INTERFACE I_TestRunner

METHOD AddTest
VAR_INPUT
    UnitTest : I_UnitTest;
END_VAR
END_METHOD

END_INTERFACE

(* stored: Version 1.1.0.1, ProductVersion 3.1.4024.11
   Itf I_TestRunner: Id {a7f355af-92fa-4f3a-9c67-696ca6bb5c15}
   Method AddTest: Id {fcbbeba9-8276-405b-893a-97438cd1031b} *)
